(* Logix 5000 project; controller SX_V040001_C001 vendor 1 type 14 code 77 rev 16.22; software revision 16.04; part 31 of 35 *)
(* tags used below, declared in another part *)
   ALL_KINDS : INT[90];
   PARAMETER : INT[501];
   pointer_param_1 : DINT;
   pointer_recipe_test : DINT;
   RECIPE_GENERAL : INT[405];
(* MainProgram, continued *)

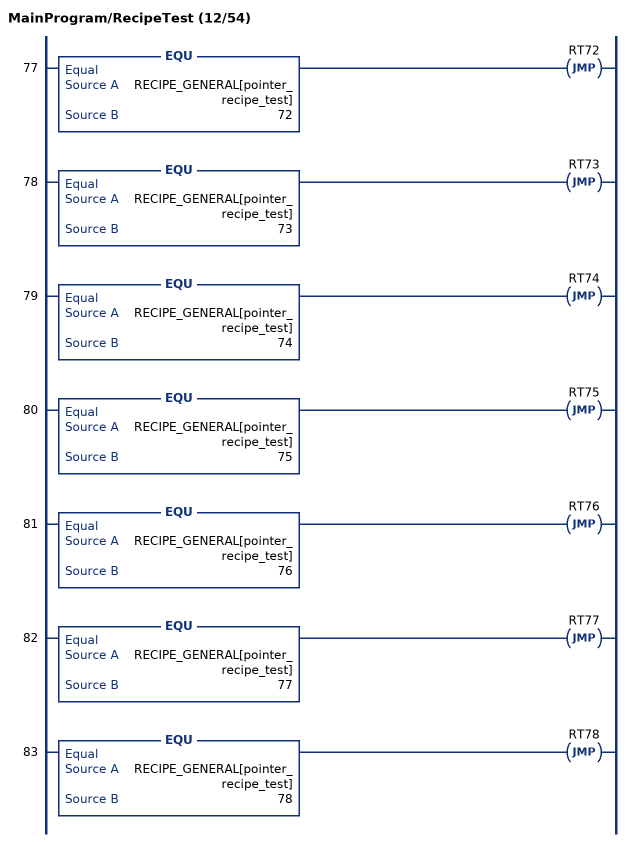
   [picture p677: MainProgram/RecipeTest rungs 77-83]
   77: EQU(RECIPE_GENERAL[pointer_recipe_test],72)JMP(RT72);
   78: EQU(RECIPE_GENERAL[pointer_recipe_test],73)JMP(RT73);
   79: EQU(RECIPE_GENERAL[pointer_recipe_test],74)JMP(RT74);
   80: EQU(RECIPE_GENERAL[pointer_recipe_test],75)JMP(RT75);
   81: EQU(RECIPE_GENERAL[pointer_recipe_test],76)JMP(RT76);
   82: EQU(RECIPE_GENERAL[pointer_recipe_test],77)JMP(RT77);
   83: EQU(RECIPE_GENERAL[pointer_recipe_test],78)JMP(RT78);
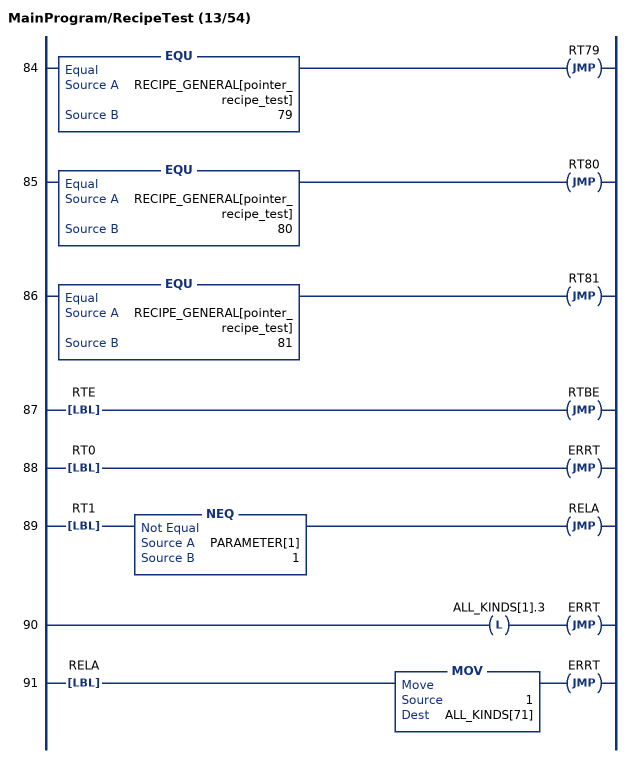
   84: EQU(RECIPE_GENERAL[pointer_recipe_test],79)JMP(RT79);
   85: EQU(RECIPE_GENERAL[pointer_recipe_test],80)JMP(RT80);
   86: EQU(RECIPE_GENERAL[pointer_recipe_test],81)JMP(RT81);
   87: LBL(RTE)JMP(RTBE);
   88: LBL(RT0)JMP(ERRT);
   89: LBL(RT1)NEQ(PARAMETER[1],1)JMP(RELA);
   90: OTL(ALL_KINDS[1].3)JMP(ERRT);
   91: LBL(RELA)MOV(1,ALL_KINDS[71])JMP(ERRT);
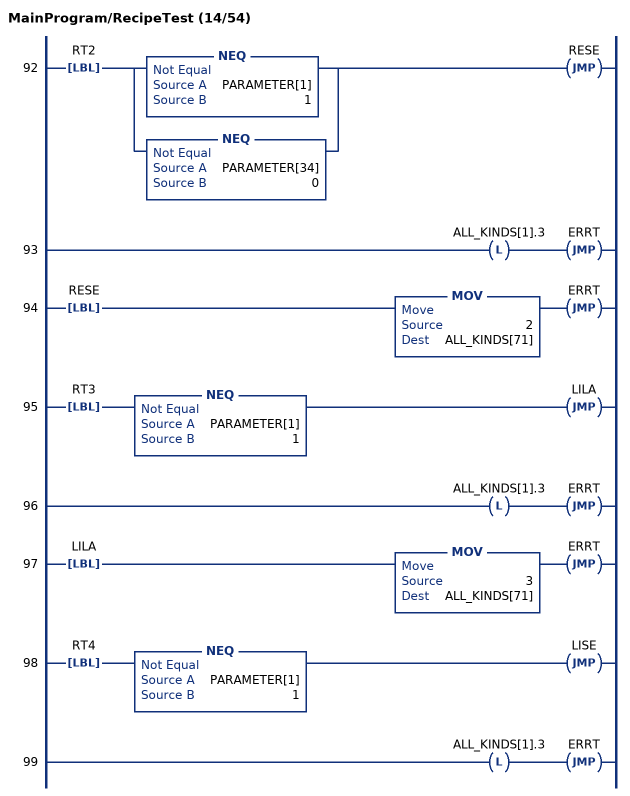
   92: LBL(RT2)[NEQ(PARAMETER[1],1) ,NEQ(PARAMETER[34],0) ]JMP(RESE);
   93: OTL(ALL_KINDS[1].3)JMP(ERRT);
   94: LBL(RESE)MOV(2,ALL_KINDS[71])JMP(ERRT);
   95: LBL(RT3)NEQ(PARAMETER[1],1)JMP(LILA);
   96: OTL(ALL_KINDS[1].3)JMP(ERRT);
   97: LBL(LILA)MOV(3,ALL_KINDS[71])JMP(ERRT);
   98: LBL(RT4)NEQ(PARAMETER[1],1)JMP(LISE);
   99: OTL(ALL_KINDS[1].3)JMP(ERRT);
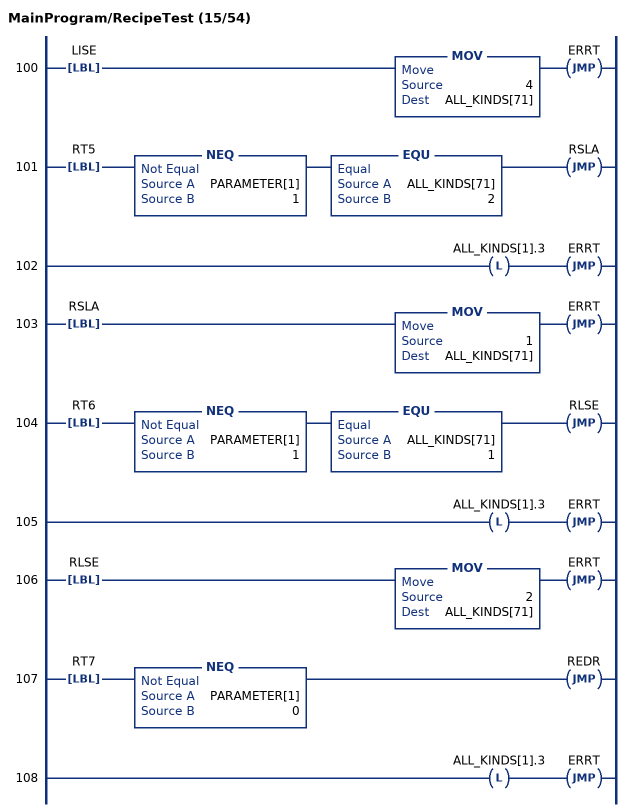
   100: LBL(LISE)MOV(4,ALL_KINDS[71])JMP(ERRT);
   101: LBL(RT5)NEQ(PARAMETER[1],1)EQU(ALL_KINDS[71],2)JMP(RSLA);
   102: OTL(ALL_KINDS[1].3)JMP(ERRT);
   103: LBL(RSLA)MOV(1,ALL_KINDS[71])JMP(ERRT);
   104: LBL(RT6)NEQ(PARAMETER[1],1)EQU(ALL_KINDS[71],1)JMP(RLSE);
   105: OTL(ALL_KINDS[1].3)JMP(ERRT);
   106: LBL(RLSE)MOV(2,ALL_KINDS[71])JMP(ERRT);
   107: LBL(RT7)NEQ(PARAMETER[1],0)JMP(REDR);
   108: OTL(ALL_KINDS[1].3)JMP(ERRT);
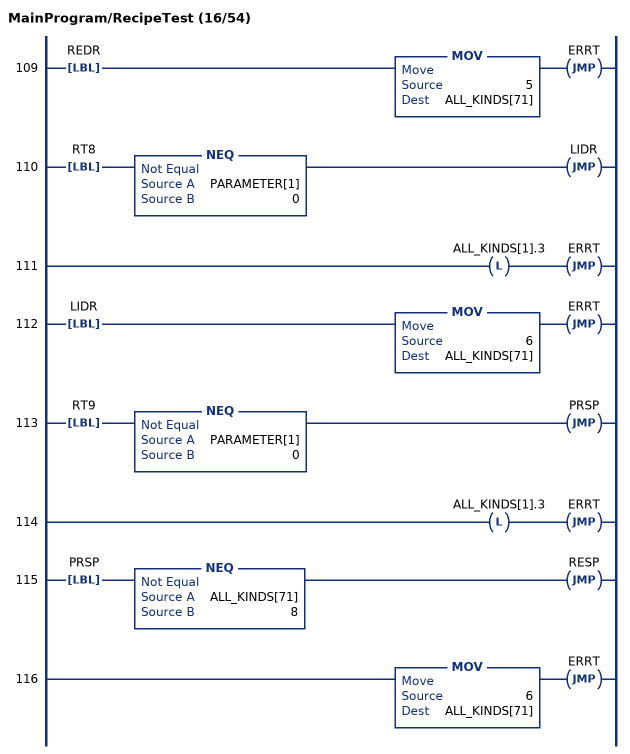
   109: LBL(REDR)MOV(5,ALL_KINDS[71])JMP(ERRT);
   110: LBL(RT8)NEQ(PARAMETER[1],0)JMP(LIDR);
   111: OTL(ALL_KINDS[1].3)JMP(ERRT);
   112: LBL(LIDR)MOV(6,ALL_KINDS[71])JMP(ERRT);
   113: LBL(RT9)NEQ(PARAMETER[1],0)JMP(PRSP);
   114: OTL(ALL_KINDS[1].3)JMP(ERRT);
   115: LBL(PRSP)NEQ(ALL_KINDS[71],8)JMP(RESP);
   116: MOV(6,ALL_KINDS[71])JMP(ERRT);
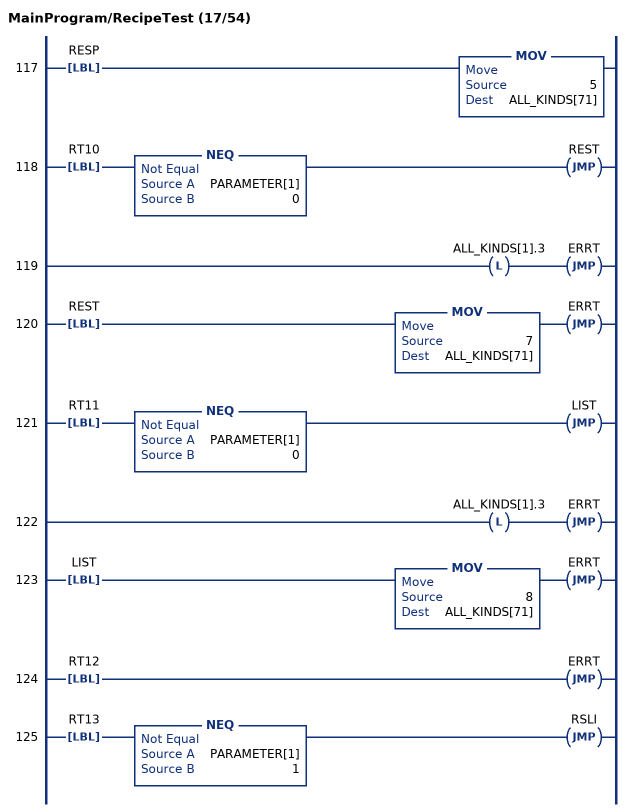
   117: LBL(RESP)MOV(5,ALL_KINDS[71]);
   118: LBL(RT10)NEQ(PARAMETER[1],0)JMP(REST);
   119: OTL(ALL_KINDS[1].3)JMP(ERRT);
   120: LBL(REST)MOV(7,ALL_KINDS[71])JMP(ERRT);
   121: LBL(RT11)NEQ(PARAMETER[1],0)JMP(LIST);
   122: OTL(ALL_KINDS[1].3)JMP(ERRT);
   123: LBL(LIST)MOV(8,ALL_KINDS[71])JMP(ERRT);
   124: LBL(RT12)JMP(ERRT);
   125: LBL(RT13)NEQ(PARAMETER[1],1)JMP(RSLI);
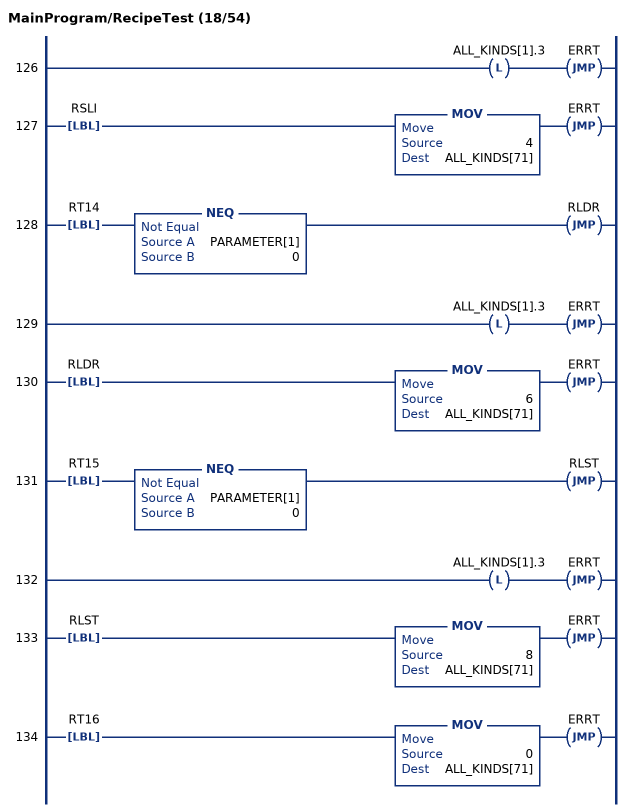
   126: OTL(ALL_KINDS[1].3)JMP(ERRT);
   127: LBL(RSLI)MOV(4,ALL_KINDS[71])JMP(ERRT);
   128: LBL(RT14)NEQ(PARAMETER[1],0)JMP(RLDR);
   129: OTL(ALL_KINDS[1].3)JMP(ERRT);
   130: LBL(RLDR)MOV(6,ALL_KINDS[71])JMP(ERRT);
   131: LBL(RT15)NEQ(PARAMETER[1],0)JMP(RLST);
   132: OTL(ALL_KINDS[1].3)JMP(ERRT);
   133: LBL(RLST)MOV(8,ALL_KINDS[71])JMP(ERRT);
   134: LBL(RT16)MOV(0,ALL_KINDS[71])JMP(ERRT);
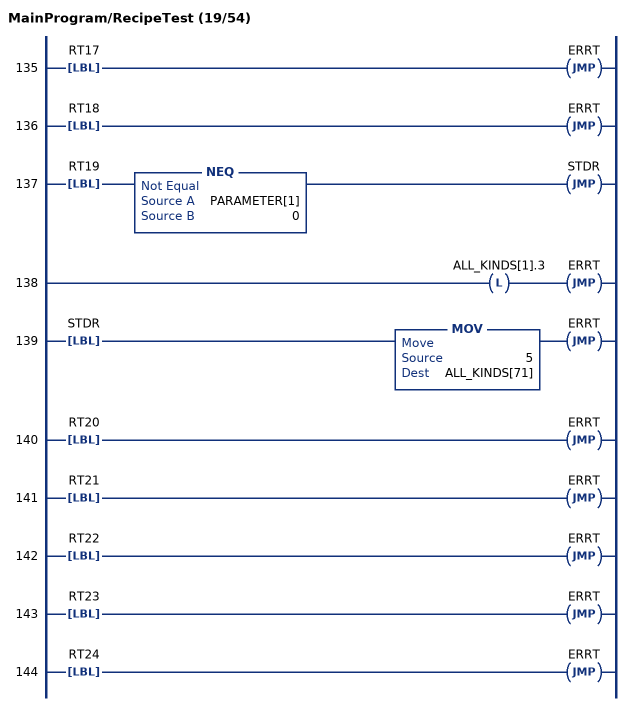
   135: LBL(RT17)JMP(ERRT);
   136: LBL(RT18)JMP(ERRT);
   137: LBL(RT19)NEQ(PARAMETER[1],0)JMP(STDR);
   138: OTL(ALL_KINDS[1].3)JMP(ERRT);
   139: LBL(STDR)MOV(5,ALL_KINDS[71])JMP(ERRT);
   140: LBL(RT20)JMP(ERRT);
   141: LBL(RT21)JMP(ERRT);
   142: LBL(RT22)JMP(ERRT);
   143: LBL(RT23)JMP(ERRT);
   144: LBL(RT24)JMP(ERRT);
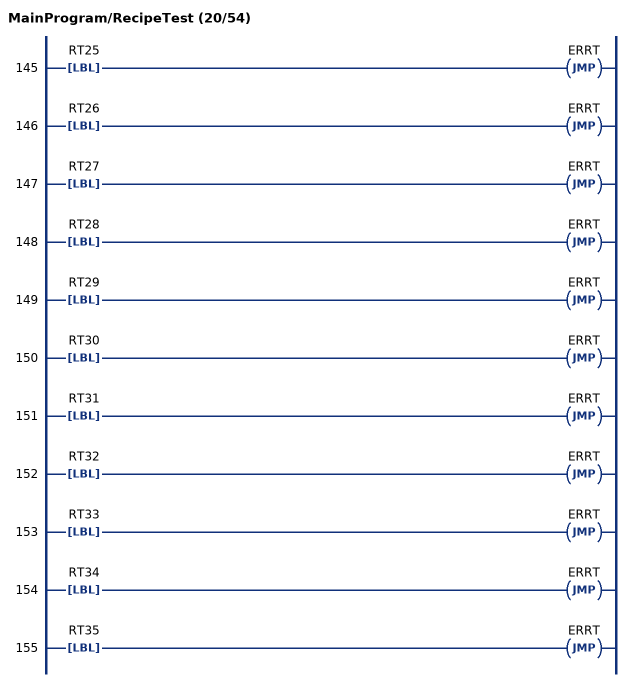
   145: LBL(RT25)JMP(ERRT);
   146: LBL(RT26)JMP(ERRT);
   147: LBL(RT27)JMP(ERRT);
   148: LBL(RT28)JMP(ERRT);
   149: LBL(RT29)JMP(ERRT);
   150: LBL(RT30)JMP(ERRT);
   151: LBL(RT31)JMP(ERRT);
   152: LBL(RT32)JMP(ERRT);
   153: LBL(RT33)JMP(ERRT);
   154: LBL(RT34)JMP(ERRT);
   155: LBL(RT35)JMP(ERRT);
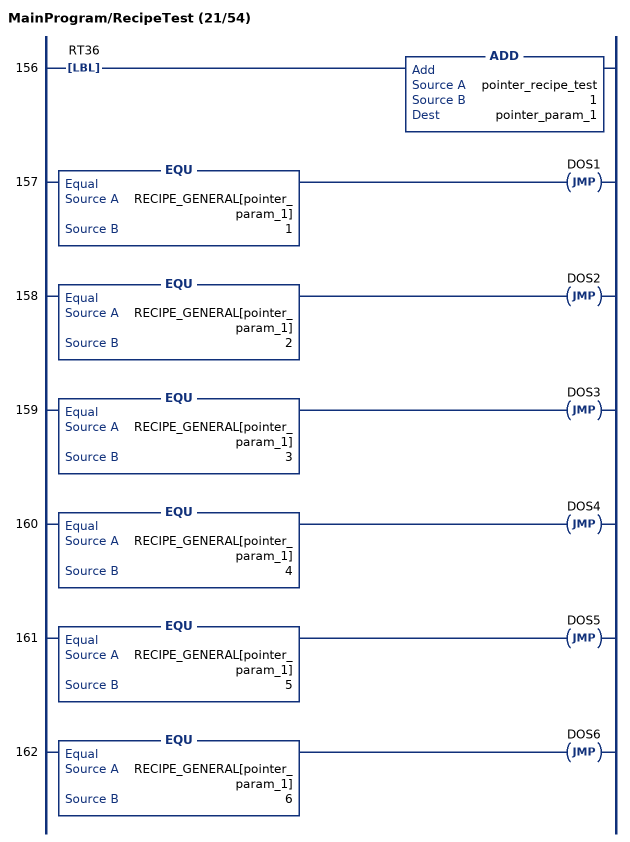
   156: LBL(RT36)ADD(pointer_recipe_test,1,pointer_param_1);
   157: EQU(RECIPE_GENERAL[pointer_param_1],1)JMP(DOS1);
   158: EQU(RECIPE_GENERAL[pointer_param_1],2)JMP(DOS2);
   159: EQU(RECIPE_GENERAL[pointer_param_1],3)JMP(DOS3);
   160: EQU(RECIPE_GENERAL[pointer_param_1],4)JMP(DOS4);
   161: EQU(RECIPE_GENERAL[pointer_param_1],5)JMP(DOS5);
   162: EQU(RECIPE_GENERAL[pointer_param_1],6)JMP(DOS6);
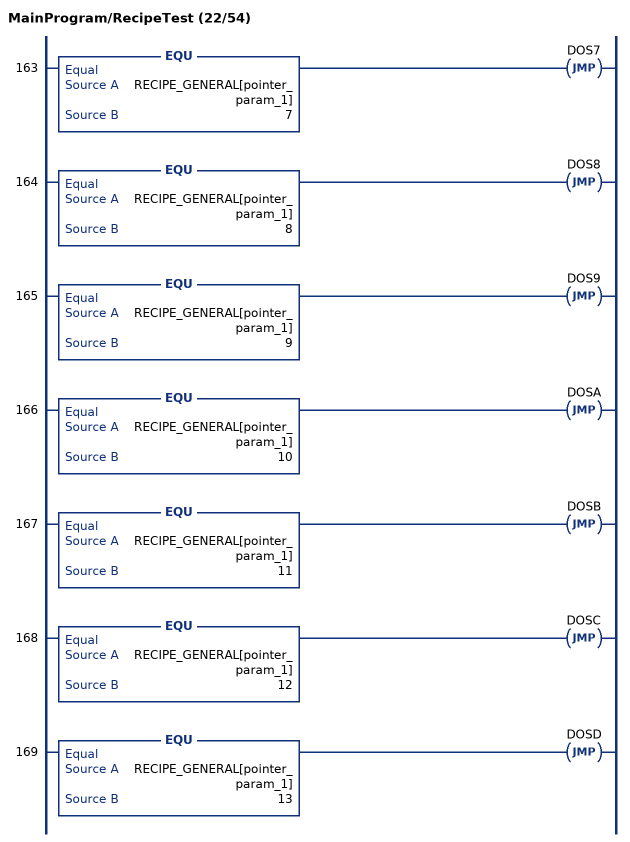
   163: EQU(RECIPE_GENERAL[pointer_param_1],7)JMP(DOS7);
   164: EQU(RECIPE_GENERAL[pointer_param_1],8)JMP(DOS8);
   165: EQU(RECIPE_GENERAL[pointer_param_1],9)JMP(DOS9);
   166: EQU(RECIPE_GENERAL[pointer_param_1],10)JMP(DOSA);
   167: EQU(RECIPE_GENERAL[pointer_param_1],11)JMP(DOSB);
   168: EQU(RECIPE_GENERAL[pointer_param_1],12)JMP(DOSC);
   169: EQU(RECIPE_GENERAL[pointer_param_1],13)JMP(DOSD);
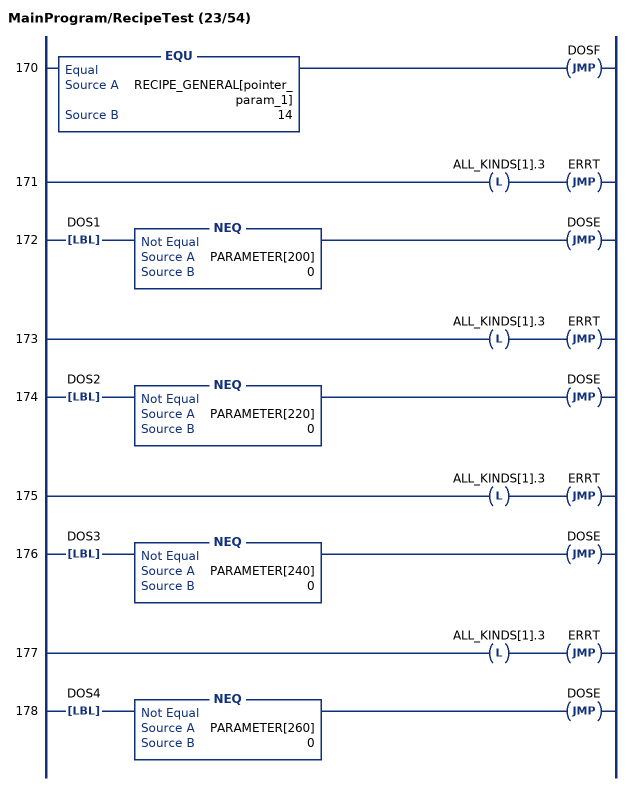
   170: EQU(RECIPE_GENERAL[pointer_param_1],14)JMP(DOSF);
   171: OTL(ALL_KINDS[1].3)JMP(ERRT);
   172: LBL(DOS1)NEQ(PARAMETER[200],0)JMP(DOSE);
   173: OTL(ALL_KINDS[1].3)JMP(ERRT);
   174: LBL(DOS2)NEQ(PARAMETER[220],0)JMP(DOSE);
   175: OTL(ALL_KINDS[1].3)JMP(ERRT);
   176: LBL(DOS3)NEQ(PARAMETER[240],0)JMP(DOSE);
   177: OTL(ALL_KINDS[1].3)JMP(ERRT);
   178: LBL(DOS4)NEQ(PARAMETER[260],0)JMP(DOSE);
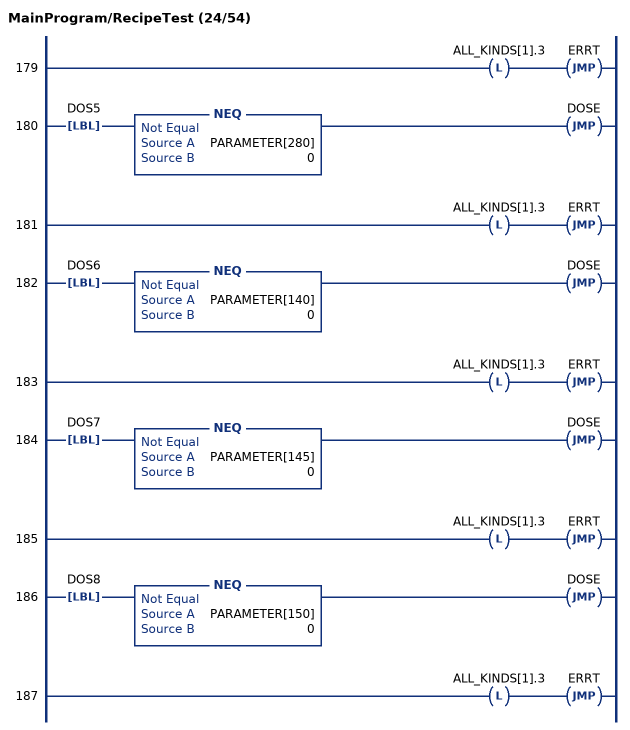
   179: OTL(ALL_KINDS[1].3)JMP(ERRT);
   180: LBL(DOS5)NEQ(PARAMETER[280],0)JMP(DOSE);
   181: OTL(ALL_KINDS[1].3)JMP(ERRT);
   182: LBL(DOS6)NEQ(PARAMETER[140],0)JMP(DOSE);
   183: OTL(ALL_KINDS[1].3)JMP(ERRT);
   184: LBL(DOS7)NEQ(PARAMETER[145],0)JMP(DOSE);
   185: OTL(ALL_KINDS[1].3)JMP(ERRT);
   186: LBL(DOS8)NEQ(PARAMETER[150],0)JMP(DOSE);
   187: OTL(ALL_KINDS[1].3)JMP(ERRT);
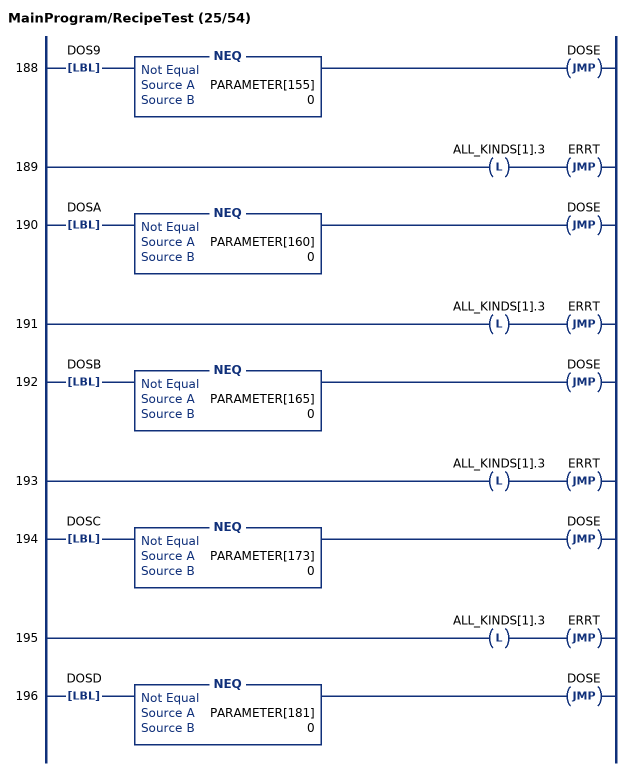
   188: LBL(DOS9)NEQ(PARAMETER[155],0)JMP(DOSE);
   189: OTL(ALL_KINDS[1].3)JMP(ERRT);
   190: LBL(DOSA)NEQ(PARAMETER[160],0)JMP(DOSE);
   191: OTL(ALL_KINDS[1].3)JMP(ERRT);
   192: LBL(DOSB)NEQ(PARAMETER[165],0)JMP(DOSE);
   193: OTL(ALL_KINDS[1].3)JMP(ERRT);
   194: LBL(DOSC)NEQ(PARAMETER[173],0)JMP(DOSE);
   195: OTL(ALL_KINDS[1].3)JMP(ERRT);
   196: LBL(DOSD)NEQ(PARAMETER[181],0)JMP(DOSE);
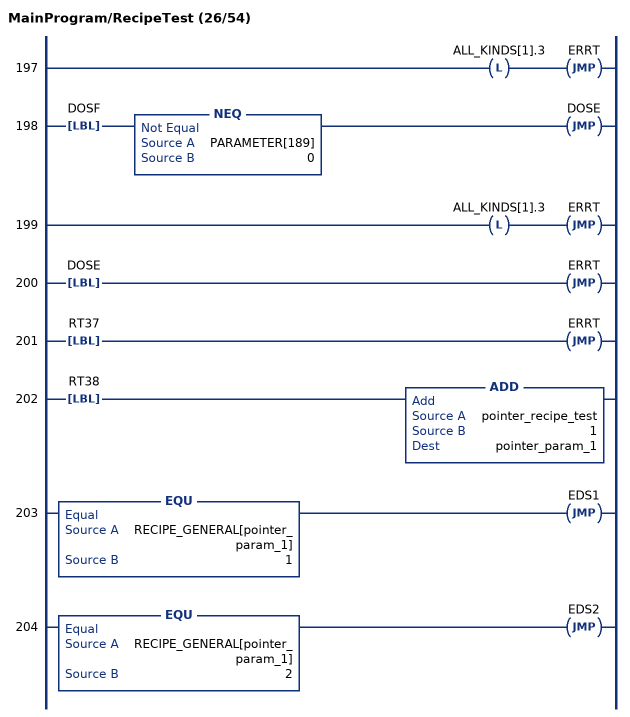
   197: OTL(ALL_KINDS[1].3)JMP(ERRT);
   198: LBL(DOSF)NEQ(PARAMETER[189],0)JMP(DOSE);
   199: OTL(ALL_KINDS[1].3)JMP(ERRT);
   200: LBL(DOSE)JMP(ERRT);
   201: LBL(RT37)JMP(ERRT);
   202: LBL(RT38)ADD(pointer_recipe_test,1,pointer_param_1);
   203: EQU(RECIPE_GENERAL[pointer_param_1],1)JMP(EDS1);
   204: EQU(RECIPE_GENERAL[pointer_param_1],2)JMP(EDS2);
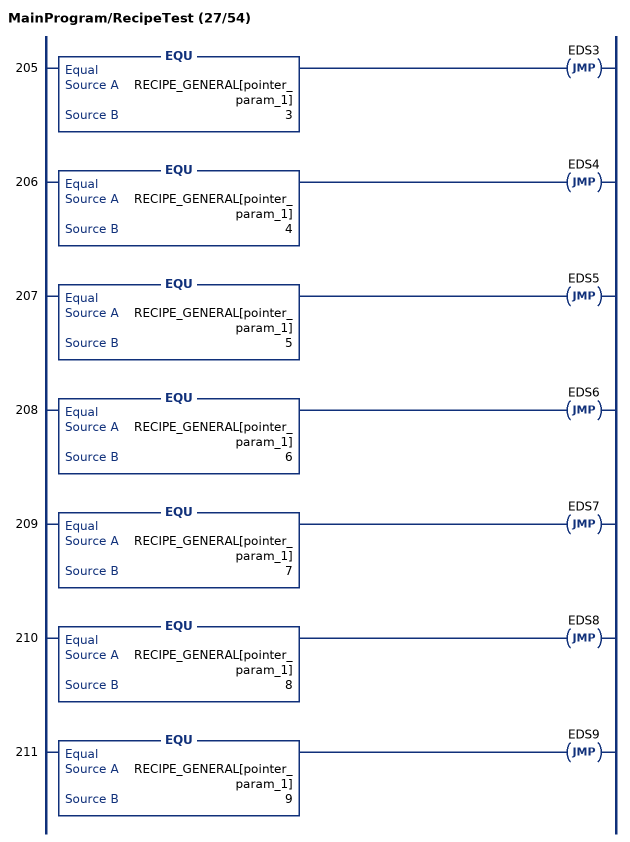
   205: EQU(RECIPE_GENERAL[pointer_param_1],3)JMP(EDS3);
   206: EQU(RECIPE_GENERAL[pointer_param_1],4)JMP(EDS4);
   207: EQU(RECIPE_GENERAL[pointer_param_1],5)JMP(EDS5);
   208: EQU(RECIPE_GENERAL[pointer_param_1],6)JMP(EDS6);
   209: EQU(RECIPE_GENERAL[pointer_param_1],7)JMP(EDS7);
   210: EQU(RECIPE_GENERAL[pointer_param_1],8)JMP(EDS8);
   211: EQU(RECIPE_GENERAL[pointer_param_1],9)JMP(EDS9);
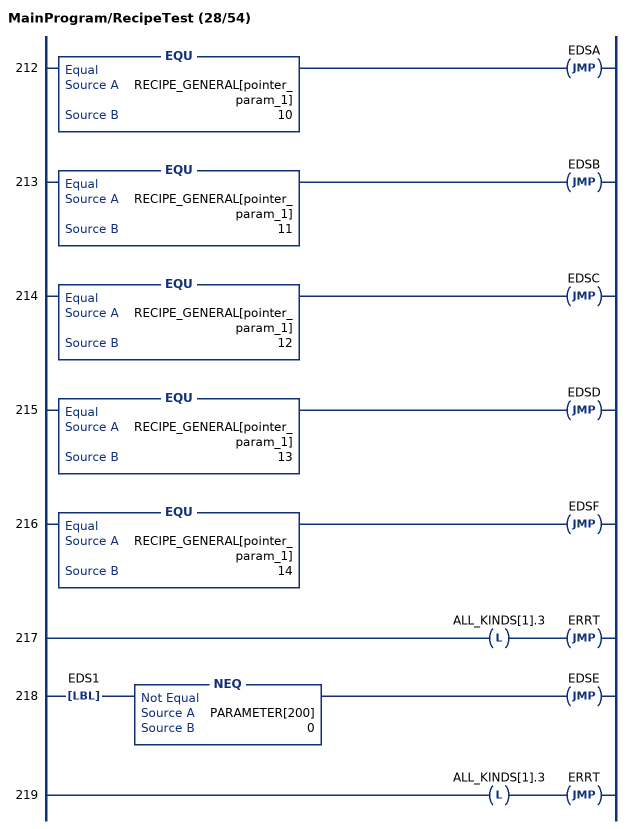
   212: EQU(RECIPE_GENERAL[pointer_param_1],10)JMP(EDSA);
   213: EQU(RECIPE_GENERAL[pointer_param_1],11)JMP(EDSB);
   214: EQU(RECIPE_GENERAL[pointer_param_1],12)JMP(EDSC);
   215: EQU(RECIPE_GENERAL[pointer_param_1],13)JMP(EDSD);
   216: EQU(RECIPE_GENERAL[pointer_param_1],14)JMP(EDSF);
   217: OTL(ALL_KINDS[1].3)JMP(ERRT);
   218: LBL(EDS1)NEQ(PARAMETER[200],0)JMP(EDSE);
   219: OTL(ALL_KINDS[1].3)JMP(ERRT);
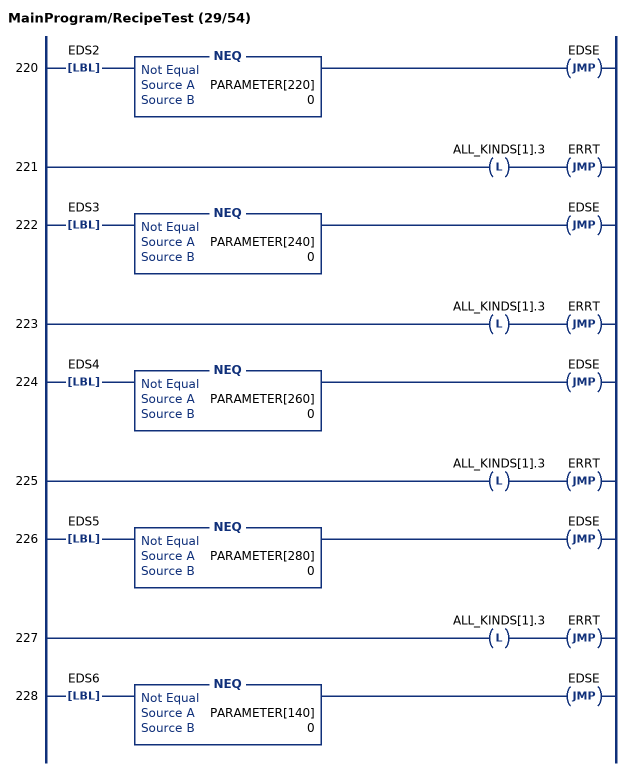
   220: LBL(EDS2)NEQ(PARAMETER[220],0)JMP(EDSE);
   221: OTL(ALL_KINDS[1].3)JMP(ERRT);
   222: LBL(EDS3)NEQ(PARAMETER[240],0)JMP(EDSE);
   223: OTL(ALL_KINDS[1].3)JMP(ERRT);
   224: LBL(EDS4)NEQ(PARAMETER[260],0)JMP(EDSE);
   225: OTL(ALL_KINDS[1].3)JMP(ERRT);
   226: LBL(EDS5)NEQ(PARAMETER[280],0)JMP(EDSE);
   227: OTL(ALL_KINDS[1].3)JMP(ERRT);
   228: LBL(EDS6)NEQ(PARAMETER[140],0)JMP(EDSE);
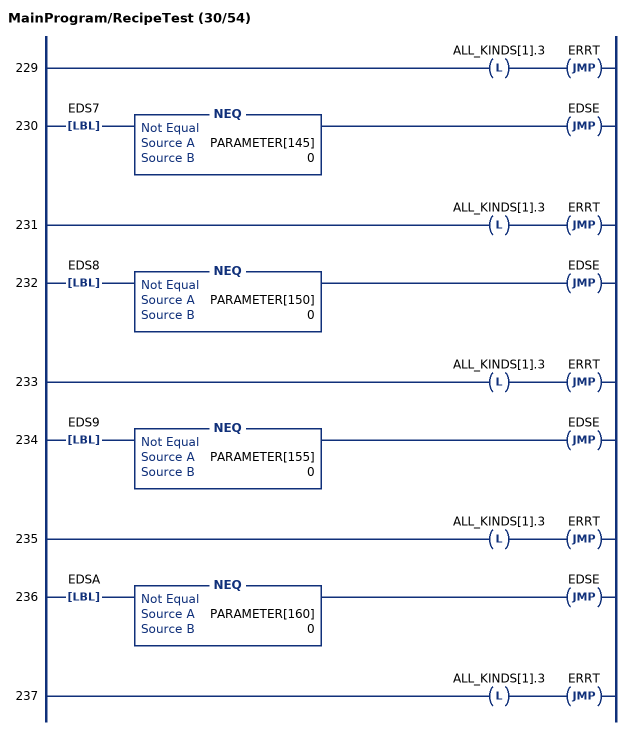
   229: OTL(ALL_KINDS[1].3)JMP(ERRT);
   230: LBL(EDS7)NEQ(PARAMETER[145],0)JMP(EDSE);
   231: OTL(ALL_KINDS[1].3)JMP(ERRT);
   232: LBL(EDS8)NEQ(PARAMETER[150],0)JMP(EDSE);
   233: OTL(ALL_KINDS[1].3)JMP(ERRT);
   234: LBL(EDS9)NEQ(PARAMETER[155],0)JMP(EDSE);
   235: OTL(ALL_KINDS[1].3)JMP(ERRT);
   236: LBL(EDSA)NEQ(PARAMETER[160],0)JMP(EDSE);
   237: OTL(ALL_KINDS[1].3)JMP(ERRT);
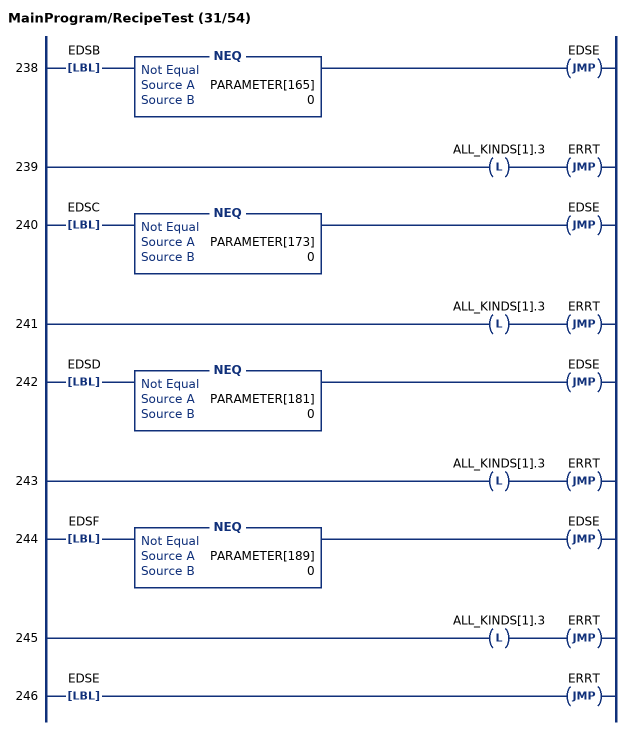
   238: LBL(EDSB)NEQ(PARAMETER[165],0)JMP(EDSE);
   239: OTL(ALL_KINDS[1].3)JMP(ERRT);
   240: LBL(EDSC)NEQ(PARAMETER[173],0)JMP(EDSE);
   241: OTL(ALL_KINDS[1].3)JMP(ERRT);
   242: LBL(EDSD)NEQ(PARAMETER[181],0)JMP(EDSE);
   243: OTL(ALL_KINDS[1].3)JMP(ERRT);
   244: LBL(EDSF)NEQ(PARAMETER[189],0)JMP(EDSE);
   245: OTL(ALL_KINDS[1].3)JMP(ERRT);
   246: LBL(EDSE)JMP(ERRT);
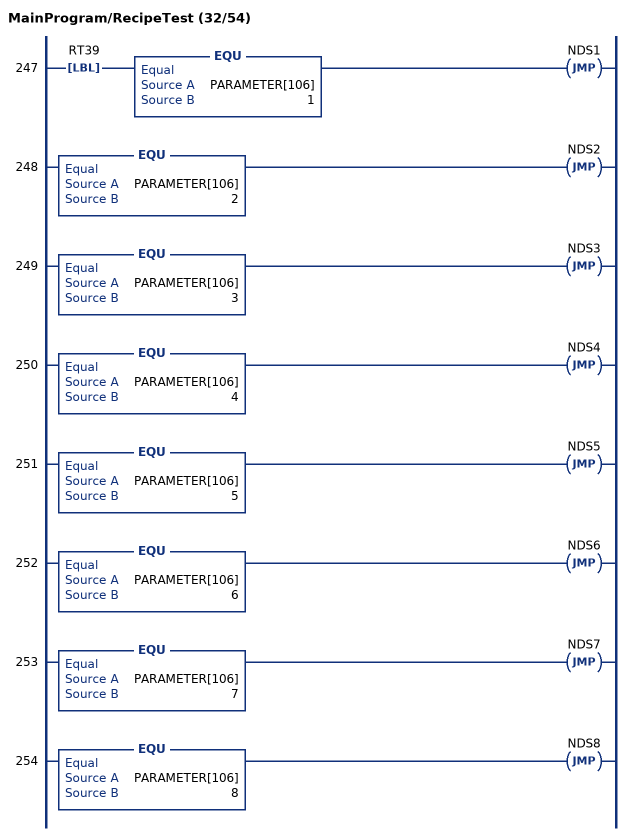
   247: LBL(RT39)EQU(PARAMETER[106],1)JMP(NDS1);
   248: EQU(PARAMETER[106],2)JMP(NDS2);
   249: EQU(PARAMETER[106],3)JMP(NDS3);
   250: EQU(PARAMETER[106],4)JMP(NDS4);
   251: EQU(PARAMETER[106],5)JMP(NDS5);
   252: EQU(PARAMETER[106],6)JMP(NDS6);
   253: EQU(PARAMETER[106],7)JMP(NDS7);
   254: EQU(PARAMETER[106],8)JMP(NDS8);
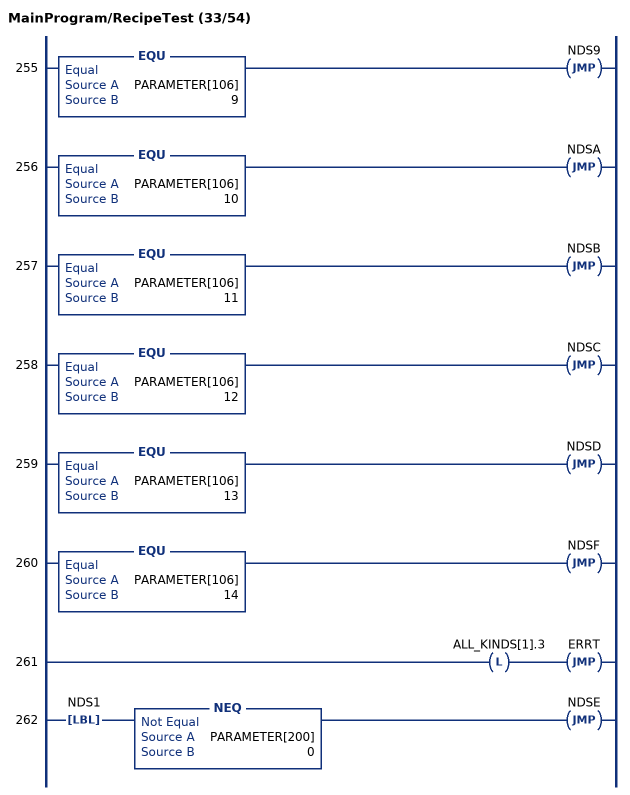
   255: EQU(PARAMETER[106],9)JMP(NDS9);
   256: EQU(PARAMETER[106],10)JMP(NDSA);
   257: EQU(PARAMETER[106],11)JMP(NDSB);
   258: EQU(PARAMETER[106],12)JMP(NDSC);
   259: EQU(PARAMETER[106],13)JMP(NDSD);
   260: EQU(PARAMETER[106],14)JMP(NDSF);
   261: OTL(ALL_KINDS[1].3)JMP(ERRT);
   262: LBL(NDS1)NEQ(PARAMETER[200],0)JMP(NDSE);
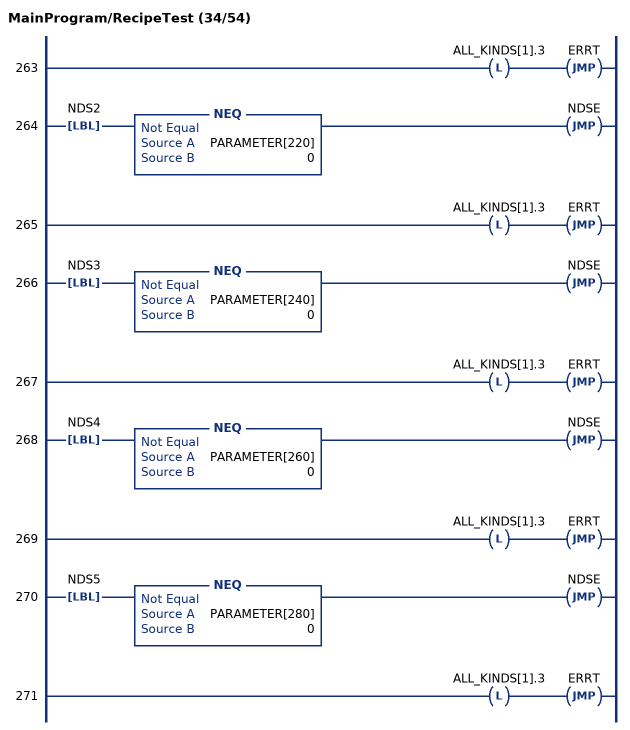
   263: OTL(ALL_KINDS[1].3)JMP(ERRT);
   264: LBL(NDS2)NEQ(PARAMETER[220],0)JMP(NDSE);
   265: OTL(ALL_KINDS[1].3)JMP(ERRT);
   266: LBL(NDS3)NEQ(PARAMETER[240],0)JMP(NDSE);
   267: OTL(ALL_KINDS[1].3)JMP(ERRT);
   268: LBL(NDS4)NEQ(PARAMETER[260],0)JMP(NDSE);
   269: OTL(ALL_KINDS[1].3)JMP(ERRT);
   270: LBL(NDS5)NEQ(PARAMETER[280],0)JMP(NDSE);
   271: OTL(ALL_KINDS[1].3)JMP(ERRT);
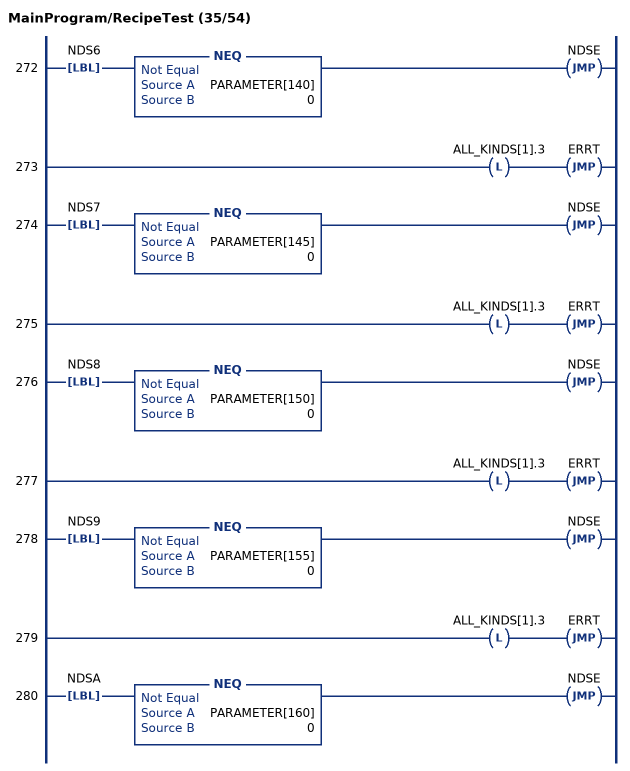
   272: LBL(NDS6)NEQ(PARAMETER[140],0)JMP(NDSE);
   273: OTL(ALL_KINDS[1].3)JMP(ERRT);
   274: LBL(NDS7)NEQ(PARAMETER[145],0)JMP(NDSE);
   275: OTL(ALL_KINDS[1].3)JMP(ERRT);
   276: LBL(NDS8)NEQ(PARAMETER[150],0)JMP(NDSE);
   277: OTL(ALL_KINDS[1].3)JMP(ERRT);
   278: LBL(NDS9)NEQ(PARAMETER[155],0)JMP(NDSE);
   279: OTL(ALL_KINDS[1].3)JMP(ERRT);
   280: LBL(NDSA)NEQ(PARAMETER[160],0)JMP(NDSE);
